// TIA Portal V20 export
TYPE "UserDiag_typeIOSystem"
TITLE = UserDiag_typeIOSystem
   STRUCT
      hardwareId { ExternalAccessible := 'False'; ExternalVisible := 'False'; ExternalWritable := 'False'} : HW_IOSYSTEM := 16#0000;   // Hardware identifier of the IO-System/DP-Mastersystem
      number { ExternalAccessible := 'False'; ExternalVisible := 'False'; ExternalWritable := 'False'} : UInt := 0;   // IO-System/DP-Mastersystem number
      error { ExternalAccessible := 'False'; ExternalVisible := 'False'; ExternalWritable := 'False'} : Bool := FALSE;   // TRUE: Error in IO-System/DP-Mastersystem
      firstDevice { ExternalAccessible := 'False'; ExternalVisible := 'False'; ExternalWritable := 'False'} : Int := 0;   // device number (index) of first device in IO System
      lastDevice { ExternalAccessible := 'False'; ExternalVisible := 'False'; ExternalWritable := 'False'} : Int := 0;   // device number (index) of last device IO System
      actualConfiguredDevices { ExternalAccessible := 'False'; ExternalVisible := 'False'; ExternalWritable := 'False'} : Int := 0;   // Number of configured devices/slaves in IO-System/DP-Mastersystem
      devices { ExternalAccessible := 'False'; ExternalVisible := 'False'; ExternalWritable := 'False'; S7_SetPoint := 'True'} : Array[1.."USERDIAG_DEVICES_PER_IO_SYSTEM_UPPER_LIM"] of "UserDiag_typeDevice";   // Device/Slave information
   END_STRUCT;
END_TYPE
